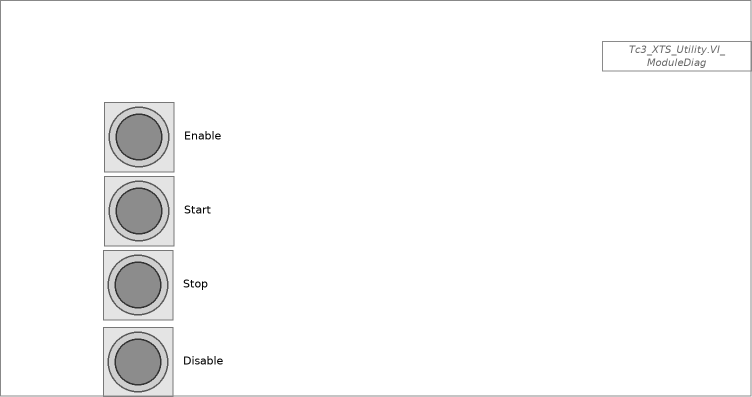
VISUALIZATION Controls  // 752x397
    PushSwitchLed (104,102 70x70), variable: GVL.XTS.Cmd.Enable, behaviour: TOGGLE, style: Switch-PushSwitchLed-Gray
    Label (181,121 150x30), "Enable"
    Label (181,195 150x30), "Start"
    PushSwitchLed (104,176 70x70), variable: GVL.XTS.Cmd.Start, behaviour: TOGGLE, style: Switch-PushSwitchLed-Gray
    Label (180,269 150x30), "Stop"
    PushSwitchLed (103,250 70x70), variable: GVL.XTS.Cmd.Stop, behaviour: TOGGLE, style: Switch-PushSwitchLed-Gray
    Label (180,346 150x30), "Disable"
    PushSwitchLed (103,327 70x70), variable: GVL.XTS.Cmd.Disable, behaviour: TOGGLE, style: Switch-PushSwitchLed-Gray
    Frame (602,41 150x30)
        shows Tc3_XTS_Utility.VI_ModuleDiag()
END_VISUALIZATION

(* stored: Version 1.1.0.1, ProductVersion 3.1.4024.12
   Visu Controls: Id {d671d5e2-5681-0862-25f9-9de6f25977db} *)
